Universal Robots PolyScope program: Dovetail_top.urp

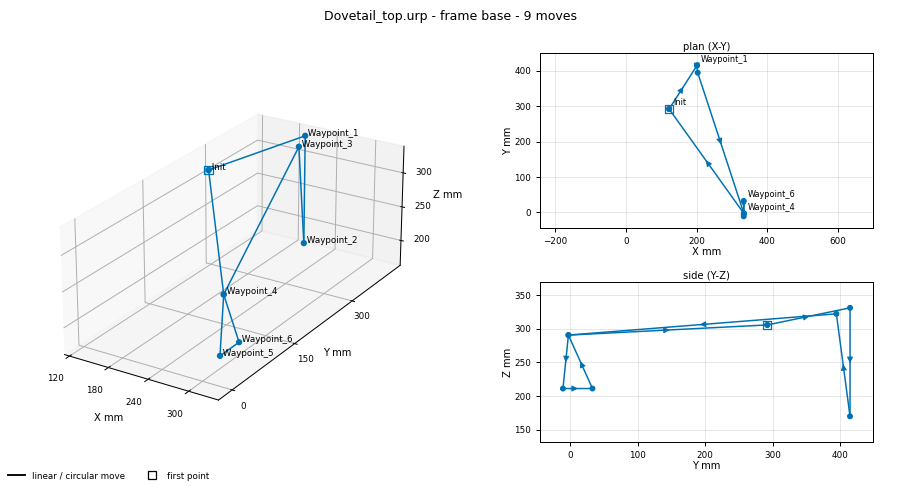
[picture p0: tool path of Dovetail_top.urp in frame base, 9 of 9 moves have a stored position in this frame; points joined in program order, loops and branches not executed]
Program Dovetail_top (installation=default directory=/programs/Mursal createdIn=5.11.11.1010533 lastSavedIn=5.11.11.1010533 robotSerialNumber=20205300864)
Calibrated DH parameters: a=[-0.000166, -0.243494, -0.153108, 0.000057, -0.000123, 0]; d=[0.151897, -1.34267, 53.988124, -52.514559, 0.085283, 0.092193]; alpha=[1.572472, -0.003756, 0.002824, 1.570807, -1.572621, 0]; deltaTheta=[0, 0.020704, 7.033215, -0.770746, 0.000004, 0]
Robot Program (runOnlyOnce=false)
  MoveL speed 250 mm/s, acceleration 1200 mm/s^2 (useActiveTCP=true) feature=Base
    Waypoint Init: TCP in base x=122.126 y=292.118 z=305.74 mm, rx=1.1346 ry=-2.9295 rz=0 rad; joints [91.639, -87.587, -91.763, -90.544, 90.033, 859.397] deg
    Waypoint Waypoint_1: TCP in base x=200.878 y=414.99 z=331.123 mm, rx=0.0832 ry=-3.1404 rz=-0.0001 rad; joints [80.689, -132.382, -22.166, -115.344, 89.821, 887.665] deg
    Waypoint Waypoint_2: TCP in base x=200.901 y=414.979 z=170.085 mm, rx=0.0831 ry=-3.1405 rz=0 rad; joints [80.576, -130.238, -70.497, -69.16, 89.918, 887.648] deg
    URCap Gripper (Robotiq_Grippers, Robotiq Inc.) dataModel(position=100.0, force=1.0, speed=0.0, positionInDouble=100.0, forceInDouble=1.0, speedInDouble=0.0, slaveIds=[9], blocking=true, robotCompliant=false)
    Waypoint Waypoint_3: TCP in base x=202.953 y=394.704 z=322.222 mm, rx=0.0453 ry=-3.0936 rz=-0.0287 rad; joints [79.305, -123.456, -40.623, -105.317, 92.75, 887.686] deg
    Waypoint Waypoint_4: TCP in base x=333.406 y=-3.075 z=290.647 mm, rx=3.1407 ry=-0.0732 rz=-0.0002 rad; joints [22.493, -91.993, -91.421, -86.491, 90.025, 655.272] deg
    Waypoint Waypoint_5: TCP in base x=332.919 y=-11.179 z=211.32 mm, rx=-3.1416 ry=0.0049 rz=-0.0001 rad; joints [21.091, -96.573, -108.555, -64.763, 90.036, 651.43] deg
    Waypoint Waypoint_6: TCP in base x=332.923 y=32.61 z=211.327 mm, rx=-3.1415 ry=0.0048 rz=-0.0001 rad; joints [28.505, -96.917, -108.158, -64.818, 90.036, 658.843] deg
    URCap Gripper (Robotiq_Grippers, Robotiq Inc.) dataModel(position=0.0, force=1.0, speed=0.0, positionInDouble=0.0, forceInDouble=1.0, speedInDouble=0.0, slaveIds=[9], blocking=true, robotCompliant=false)
    Waypoint Waypoint_4: TCP in base x=333.406 y=-3.075 z=290.647 mm, rx=3.1407 ry=-0.0732 rz=-0.0002 rad; joints [22.493, -91.993, -91.421, -86.491, 90.025, 655.272] deg
    Waypoint Init: TCP in base x=122.126 y=292.118 z=305.74 mm, rx=1.1346 ry=-2.9295 rz=0 rad; joints [91.639, -87.587, -91.763, -90.544, 90.033, 859.397] deg
